Staubli VAL3: ContorlLight.pgx

program ContorlLight()
begin
  //

  while !bExit
    //红灯
    if PublicData:sStatus=="stop"
      IO:dOut["dOut2"]=true
      IO:dOut["dOut3"]=false
      IO:dOut["dOut4"]=false
    elseIf PublicData:sStatus=="pause"
      IO:dOut["dOut2"]=false
      IO:dOut["dOut3"]=false
      IO:dOut["dOut4"]=true
    elseIf PublicData:sStatus=="run"
      IO:dOut["dOut2"]=false
      IO:dOut["dOut3"]=true
      IO:dOut["dOut4"]=false
    endIf
    delay(0)
  endWhile

end
